{attribute 'qualified_only'}
{attribute 'strict'}
TYPE Positions :
(
	First := 180,
	Second:=148,
	Third:=116,
	Forth:=84
);
END_TYPE

(* stored: Version 1.1.0.1, ProductVersion 3.1.4024.3
   DUT Positions: Id {0428c303-5827-472d-915e-9f54d811f361} *)
